FUNCTION_BLOCK PT1T2_Prozess
VAR_INPUT
	u :			REAL;
	Modus :		System_Modus_Enum;
	Param :		PT1T2_Parameter_Strukt;
	T :			REAL;
END_VAR
VAR_OUTPUT
	y :			REAL;
END_VAR
VAR
	alpha1 :	REAL;
	alpha2 :	REAL;
	a1 :		REAL;
	a2 :		REAL;
	b0 :		REAL;
	b1 :		REAL;
	b2 :		REAL;
	
	ym :		REAL;
	ymm :		REAL;
END_VAR

CASE Modus OF
	System_Modus_Enum.System_Init:
	alpha1 := T + Param.T1;
	alpha2 := T + Param.T2;
	a1 := 1;
	a2 := 2;
	b0 := (Param.K*T*T)/(alpha1*alpha2);
	a1 := -((Param.T1/alpha1)+(Param.T2/alpha2));
	a2 := (Param.T1*Param.T2)/(alpha1*alpha2);
	y := 0;
	ym := 0;
	ymm := 0;
	;
	System_Modus_Enum.System_Run:
	y := -a1 * ym - a2 *ymm + b0 * u;
	ymm := ym;
	ym := y;
	;
END_CASE

END_FUNCTION_BLOCK

(* stored: Version 1.1.0.1, ProductVersion 3.1.4024.13
   POU PT1T2_Prozess: Id {e56b3e77-136a-481d-9d19-c322548e5a49}, SpecialFunc None *)
